// TIA Portal project "shift_registers" (V14)
// Cf. https://www.plctalk.net/qanda/showthread.php?t=128167

(* hardware
DEVICE "S7-1200 station_1"  S7-1200 Station
   slot 0: "Rack_0"  Rack  V1.0
   slot 1: "PLC_1"  CPU 1214C DC/DC/DC  6ES7 214-1AG40-0XB0  V4.2
DEVICE "HMI_1"  KTP700 Basic PN Portrait
   slot 0: "KTP700 Basic PN Portrait"  KTP700 Basic PN Portrait  6AV2 123-2GB03-0AX0  14.0.0.0
   slot 1: "HMI_RT_1"  KTP700 Basic PN Portrait  6AV2 123-2GB03-0AX0  14.0.0.0
   slot 5: "HMI_1.IE_CP_1"  PROFINET Interface  14.0.0.0
      slot 1: "PROFINET Interface_1"  PROFINET Interface
         slot 1: "Port_1"  Port
*)

// ===== PLC "PLC_1"  CPU 1214C DC/DC/DC =====

VAR_GLOBAL   // PLC tag table "Default tag table"
   "new_product_prox_input" AT %M0.6 : Bool;
   "HMI_ingest_input" AT %M0.7 : Bool;
   "HMI_target_line_input" AT %MW104 : Int;
   "HMI_target_pitch_input" AT %MW106 : Int;
   "Pause" AT %M1.1 : Bool;
   "current_pitch" AT %MW108 : Int;
   "valve_1" AT %M2.0 : Bool;
   "valve_2" AT %M2.1 : Bool;
   "valve_3" AT %M2.2 : Bool;
   "valve_4" AT %M2.3 : Bool;
   "valve_5" AT %M2.4 : Bool;
   "valve_6" AT %M2.5 : Bool;
   "Run" AT %M0.0 : Bool;
   "HMI_start_input" AT %M0.4 : Bool;
   "HMI_stop_input" AT %M0.5 : Bool;
   "pitch_prox_input" AT %M1.0 : Bool;
   "ingest_new" AT %M0.1 : Bool;
   "target_line" AT %MW100 : Int;
   "target_pitch" AT %MW102 : Int;
   "pitch_pulse" AT %M0.2 : Bool;
   "pitch_pulse_M" AT %M1.2 : Bool;
   "run_simulator" AT %M1.3 : Bool;
END_VAR

DATA_BLOCK "InputMap_DB"   // DB1
{ S7_Optimized_Access := 'TRUE' }
VERSION : 0.1
// stored: InstanceOfName InputMap
"InputMap"
BEGIN
END_DATA_BLOCK

DATA_BLOCK "LineValve_DB_1"   // DB2
{ S7_Optimized_Access := 'TRUE' }
VERSION : 0.1
// stored: InstanceOfName LineValve
"LineValve"
BEGIN
END_DATA_BLOCK

DATA_BLOCK "FIFO_BITS"   // DB3
{ S7_Optimized_Access := 'TRUE' }
VERSION : 0.1
   VAR
      fifo_bits : Array[0..511] of Byte;
   END_VAR
BEGIN
END_DATA_BLOCK

DATA_BLOCK "LineValve_DB_2"   // DB4
{ S7_Optimized_Access := 'TRUE' }
VERSION : 0.1
// stored: InstanceOfName LineValve
"LineValve"
BEGIN
END_DATA_BLOCK

DATA_BLOCK "LineValve_DB_3"   // DB5
{ S7_Optimized_Access := 'TRUE' }
VERSION : 0.1
// stored: InstanceOfName LineValve
"LineValve"
BEGIN
END_DATA_BLOCK

DATA_BLOCK "LineValve_DB_4"   // DB6
{ S7_Optimized_Access := 'TRUE' }
VERSION : 0.1
// stored: InstanceOfName LineValve
"LineValve"
BEGIN
END_DATA_BLOCK

DATA_BLOCK "LineValve_DB_5"   // DB7
{ S7_Optimized_Access := 'TRUE' }
VERSION : 0.1
// stored: InstanceOfName LineValve
"LineValve"
BEGIN
END_DATA_BLOCK

DATA_BLOCK "LineValve_DB_6"   // DB8
{ S7_Optimized_Access := 'TRUE' }
VERSION : 0.1
// stored: InstanceOfName LineValve
"LineValve"
BEGIN
END_DATA_BLOCK

DATA_BLOCK "Simulator_DB"   // DB9
{ S7_Optimized_Access := 'TRUE' }
VERSION : 0.1
// stored: InstanceOfName Simulator
"Simulator"
BEGIN
END_DATA_BLOCK

FUNCTION_BLOCK "InputMap"   // FB1, LAD
TITLE = Process HMI and sensor inputs
{ S7_Optimized_Access := 'TRUE' }
VERSION : 0.1
// N.B. new_product_prox_input probably needs a debounce for both 0-to-1 and 1-to-0 transitons; same for the pitch input
   VAR_INPUT
      new_product_prox_input : Bool;
      pitch_input : Bool;
   END_VAR
   VAR_OUTPUT
      Run_output : Bool;
      Pause_output : Bool;
      Ingest_output : Bool;
      target_line_output : Int;
      target_pitch_output : Int;
      pitch_pulse_output : Bool;
   END_VAR
   VAR_IN_OUT
      HMI_start_InOut : Bool;
      HMI_stop_InOut : Bool;
      HMI_ingest_InOut : Bool;
      HMI_target_line_InOut : Int;
      HMI_target_pitch_InOut : Int;
   END_VAR
   VAR
      Run : Bool;
      Pause : Bool;
      Ingest : Bool;
      new_product_prox_M : Bool;
      ingest_M : Bool;
      HMI_Line_pitch_offsets : Array[0..6] of Int;
   END_VAR
   VAR_TEMP   // added for the SCL form of the ladder/FBD networks
      _w1 : Bool;
      _w2 : Bool;
      _w3 : Bool;
   END_VAR
   // HMI_Line_pitch_offsets[1] := 4;
   // HMI_Line_pitch_offsets[2] := 8;
   // HMI_Line_pitch_offsets[3] := 12;
   // HMI_Line_pitch_offsets[4] := 16;
   // HMI_Line_pitch_offsets[5] := 20;
   // HMI_Line_pitch_offsets[6] := 24;
   // HMI_Line_pitch_offsets[0] := 0;
BEGIN

REGION Network 1: Process Start/Stop from HMI to Run
   // Also Reset HMI-driven Start/Stop to avoid anomalies if HMI does not return either of those momentaries to 0 ("set and forget")
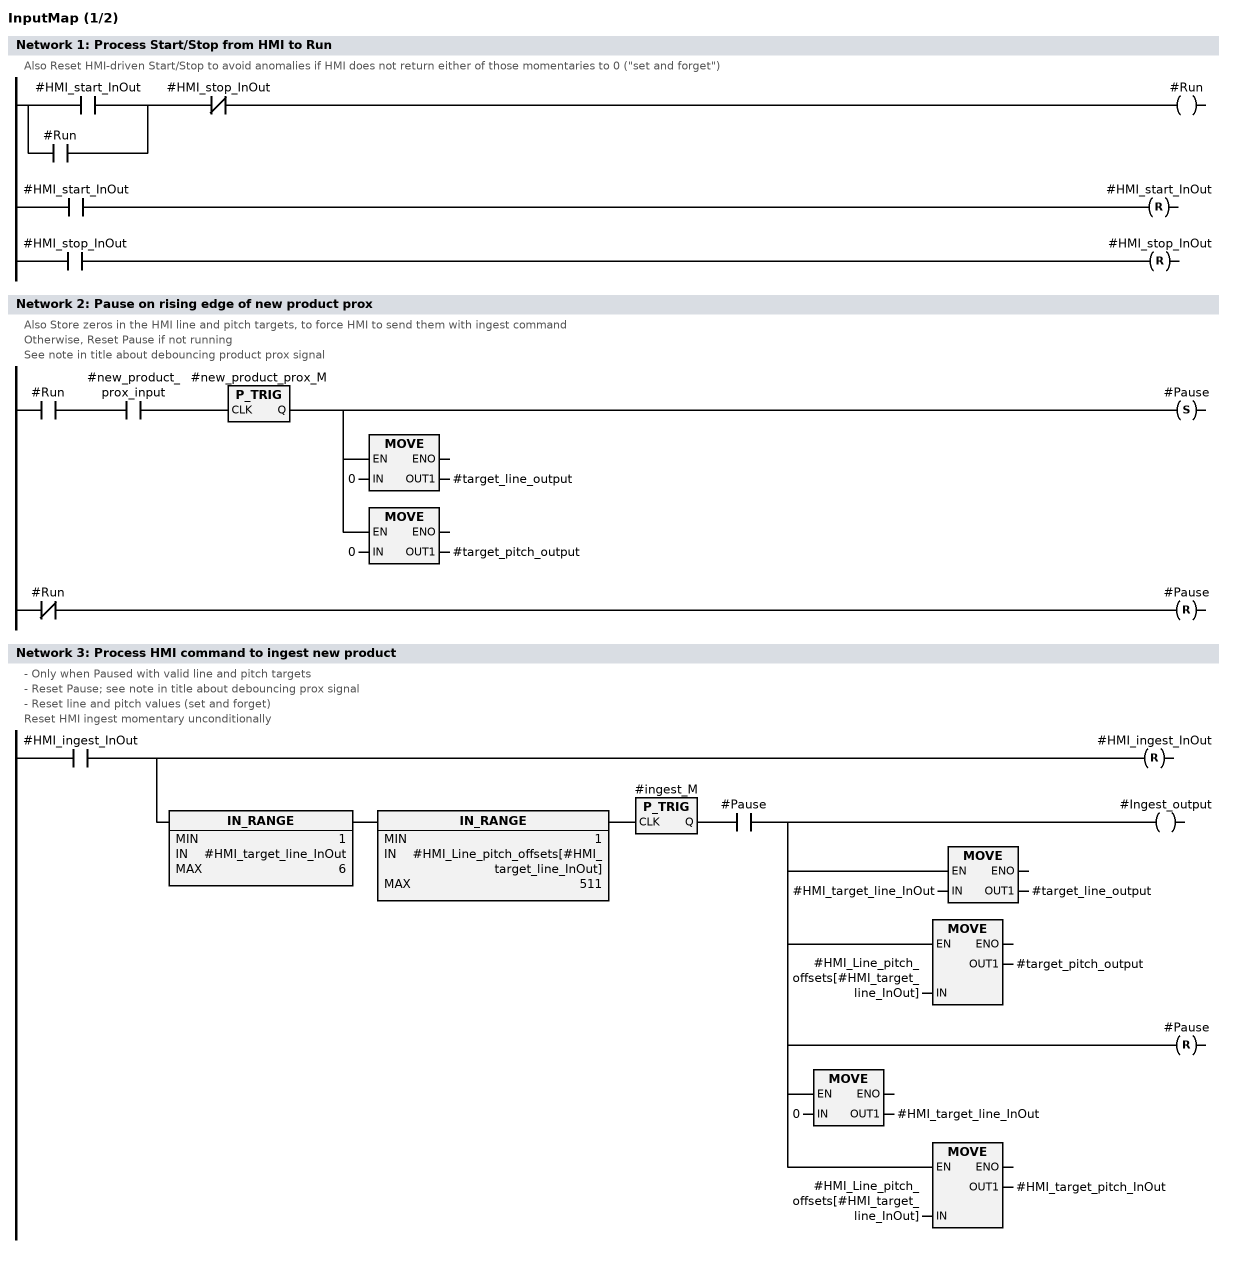
   RUNG wire#powerrail
      Contact( #HMI_start_InOut )
      wire#w1
      I_Contact( #HMI_stop_InOut )
      Coil( #Run )
   END_RUNG
   RUNG wire#powerrail
      Contact( #Run )
   END_RUNG wire#w1
   RUNG wire#powerrail
      Contact( #HMI_start_InOut )
      R_Coil( #HMI_start_InOut )
   END_RUNG
   RUNG wire#powerrail
      Contact( #HMI_stop_InOut )
      R_Coil( #HMI_stop_InOut )
   END_RUNG
   // the same network as SCL:
   #Run := (#HMI_start_InOut OR #Run) AND NOT #HMI_stop_InOut;
   IF #HMI_start_InOut THEN #HMI_start_InOut := FALSE; END_IF;
   IF #HMI_stop_InOut THEN #HMI_stop_InOut := FALSE; END_IF;
END_REGION

REGION Network 2: Pause on rising edge of new product prox
   // Also Store zeros in the HMI line and pitch targets, to force HMI to send them with ingest command
   // Otherwise, Reset Pause if not running
   // See note in title about debouncing product prox signal
   RUNG wire#powerrail
      Contact( #Run )
      Contact( #new_product_prox_input )
      P_Trig( #new_product_prox_M )
      wire#w1
      S_Coil( #Pause )
   END_RUNG
   RUNG wire#w1
      Move(in := 0, out1 => #target_line_output)
   END_RUNG
   RUNG wire#w1
      Move(in := 0, out1 => #target_pitch_output)
   END_RUNG
   RUNG wire#powerrail
      I_Contact( #Run )
      R_Coil( #Pause )
   END_RUNG
   // the same network as SCL:
   #_w1 := #Run AND #new_product_prox_input;
   #_w2 := #_w1 AND NOT #new_product_prox_M;   // rising edge
   #new_product_prox_M := #_w1;
   IF #_w2 THEN
       #Pause := TRUE;
       #target_line_output := 0;
       #target_pitch_output := 0;
   END_IF;
   IF NOT #Run THEN #Pause := FALSE; END_IF;
END_REGION

REGION Network 3: Process HMI command to ingest new product
   // - Only when Paused with valid line and pitch targets
   // - Reset Pause; see note in title about debouncing prox signal
   // - Reset line and pitch values (set and forget)
   // Reset HMI ingest momentary unconditionally
   RUNG wire#powerrail
      Contact( #HMI_ingest_InOut )
      wire#w1
      R_Coil( #HMI_ingest_InOut )
   END_RUNG
   RUNG wire#w1
      { S7_Templates := "SrcType := Int" } InRange(min := 1, in := #HMI_target_line_InOut, max := 6)
      { S7_Templates := "SrcType := Int" } InRange(min := 1, in := #HMI_Line_pitch_offsets[#HMI_target_line_InOut], max := 511)
      P_Trig( #ingest_M )
      Contact( #Pause )
      wire#w2
      Coil( #Ingest_output )
   END_RUNG
   RUNG wire#w2
      Move(in := #HMI_target_line_InOut, out1 => #target_line_output)
   END_RUNG
   RUNG wire#w2
      Move(in := #HMI_Line_pitch_offsets[#HMI_target_line_InOut], out1 => #target_pitch_output)
   END_RUNG
   RUNG wire#w2
      R_Coil( #Pause )
   END_RUNG
   RUNG wire#w2
      Move(in := 0, out1 => #HMI_target_line_InOut)
   END_RUNG
   RUNG wire#w2
      Move(in := #HMI_Line_pitch_offsets[#HMI_target_line_InOut], out1 => #HMI_target_pitch_InOut)
   END_RUNG
   // the same network as SCL:
   #_w1 := #HMI_ingest_InOut;
   IF #_w1 THEN #HMI_ingest_InOut := FALSE; END_IF;
   #_w2 := #_w1 AND (1 <= #HMI_target_line_InOut) AND (#HMI_target_line_InOut <= 6) AND (1 <= #HMI_Line_pitch_offsets[#HMI_target_line_InOut]) AND (#HMI_Line_pitch_offsets[#HMI_target_line_InOut] <= 511);
   #_w3 := #_w2 AND NOT #ingest_M;   // rising edge
   #ingest_M := #_w2;
   #Ingest_output := #_w3 AND #Pause;
   IF #Ingest_output THEN
       #target_line_output := #HMI_target_line_InOut;
       #target_pitch_output := #HMI_Line_pitch_offsets[#HMI_target_line_InOut];
       #Pause := FALSE;
       #HMI_target_line_InOut := 0;
       #HMI_target_pitch_InOut := #HMI_Line_pitch_offsets[#HMI_target_line_InOut];
   END_IF;
END_REGION

REGION Network 4: Push values to remaining outputs
   // - A debounce circuit for the pitch input might not go amiss here
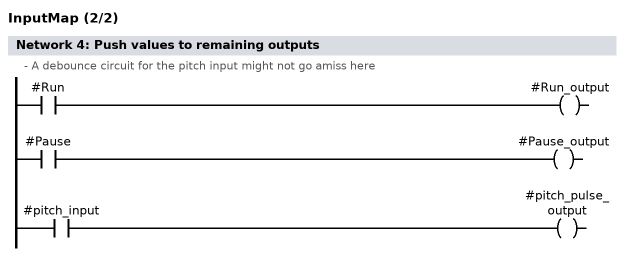
   RUNG wire#powerrail
      Contact( #Run )
      Coil( #Run_output )
   END_RUNG
   RUNG wire#powerrail
      Contact( #Pause )
      Coil( #Pause_output )
   END_RUNG
   RUNG wire#powerrail
      Contact( #pitch_input )
      Coil( #pitch_pulse_output )
   END_RUNG
   // the same network as SCL:
   #Run_output := #Run;
   #Pause_output := #Pause;
   #pitch_pulse_output := #pitch_input;
END_REGION
END_FUNCTION_BLOCK

FUNCTION_BLOCK "LineValve"   // FB2, LAD
TITLE = Process inputs for one Line-valve
{ S7_Optimized_Access := 'TRUE' }
VERSION : 0.1
// - Operate valve
// - Set up to ingest  three bits on ingest_pulse directed at this Line
// - Ingest those three bits on successive pitch rising edges
   VAR_INPUT
      target_line : Int;   // Line to ingest target_pitch if ingest_pulse is 0
      target_pitch : Int;   // Pitch offset of target_line if ingest_pulse is 0
      this_line : Int;   // Which Line this is
      current_pitch : Int;   // Conveyor start pitch offset into fifo_bits
      pitch_pulse : Bool;   // Pitch detection
   END_VAR
   VAR_OUTPUT
      operate_valve : Bool;   // Valve to direct product to ths Line
   END_VAR
   VAR_IN_OUT
      ingest_pulse : Bool;   // Bit commanding target_line to ingest target_pitch
      fifo_bits : Array[0..511] of Byte;   // Byte array containing product flag for all lines
   END_VAR
   VAR
      bits_to_ingest : Int;   // Remaining bits to ingest on pitch_pulse rising edges
      saved_pitch_offset : Int;   // Pitch offset from start of conveyor to this line's valve
      ingest_M : Bool;
   END_VAR
   VAR_TEMP
      this_bit_at_X7 : Byte;
      future_pitch : Int;
      this_bit : Int;
   END_VAR
   VAR CONSTANT
      pctX7 : Int := 2#10000000;
   END_VAR
   VAR_TEMP   // added for the SCL form of the ladder/FBD networks
      _w1 : Bool;
      _w2 : Bool;
   END_VAR
BEGIN

REGION Network 1: Operate valve when modeled product destined for this Line is near its Valve
   // Detect when the bit for this Line in Byte fifo_bits[current_pitch] is 1
   // - Bits in the static FIFO are cleared in Main [OB1] when current_pitch increments at pitch rising edge
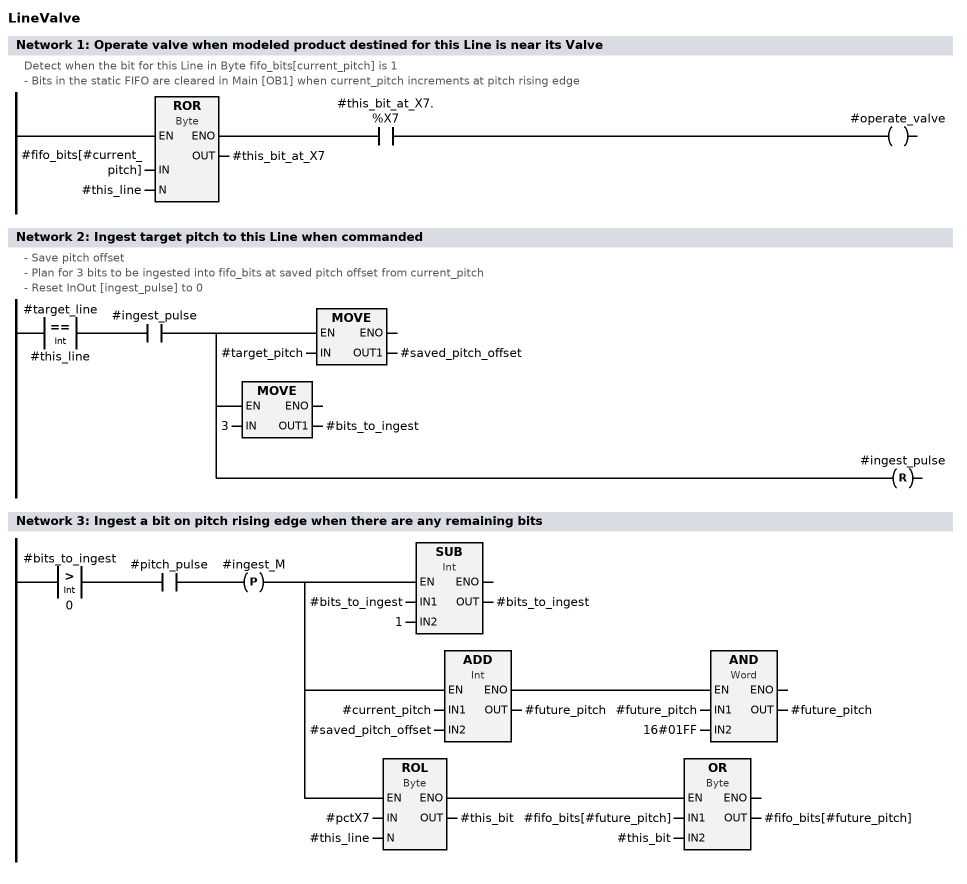
   #this_bit_at_X7 := ROR(IN := #fifo_bits[#current_pitch], N := #this_line);
   #operate_valve := #this_bit_at_X7.%X7;
END_REGION

REGION Network 2: Ingest target pitch to this Line when commanded
   // - Save pitch offset
   // - Plan for 3 bits to be ingested into fifo_bits at saved pitch offset from current_pitch
   // - Reset InOut [ingest_pulse] to 0
   RUNG wire#powerrail
      { S7_Templates := "SrcType := Int" } EQ_Contact(in1 := #target_line, in2 := #this_line)
      Contact( #ingest_pulse )
      wire#w1
      Move(in := #target_pitch, out1 => #saved_pitch_offset)
   END_RUNG
   RUNG wire#w1
      Move(in := 3, out1 => #bits_to_ingest)
   END_RUNG
   RUNG wire#w1
      R_Coil( #ingest_pulse )
   END_RUNG
   // the same network as SCL:
   IF (#target_line = #this_line) AND #ingest_pulse THEN
       #saved_pitch_offset := #target_pitch;
       #bits_to_ingest := 3;
       #ingest_pulse := FALSE;
   END_IF;
END_REGION

REGION Network 3: Ingest a bit on pitch rising edge when there are any remaining bits
   // no checked SCL form for this network; see the picture
END_REGION
END_FUNCTION_BLOCK

FUNCTION_BLOCK "Simulator"   // FB3, LAD
TITLE = Model/simulate synthetic inputs from HMI and physical sensors (pitch and new product proxes)
{ S7_Optimized_Access := 'TRUE' }
VERSION : 0.1
   VAR_INPUT
      Run_this_sim_Input : Bool;
      Run_Input : Bool;
      Pause_Input : Bool;
   END_VAR
   VAR_IN_OUT
      pitch_prox_InOut : Bool;
      new_product_prox_InOut : Bool;
   END_VAR
   VAR
      time_status : Int;
      time_dtl : DTL;
      next_target_line : Int;
      IEC_prox_delay : IEC_TIMER;
      second : USInt;
      nanosecond : UDInt;
      two_second_M : Bool;
      prox_pulse : Bool;
      new_product_prox_delay_count : Int;
   END_VAR
   VAR_TEMP   // added for the SCL form of the ladder/FBD networks
      _w1 : Bool;
      _w2 : Bool;
      _w3 : Bool;
   END_VAR
BEGIN

REGION Network 1: RETurn if simulator is not to be run
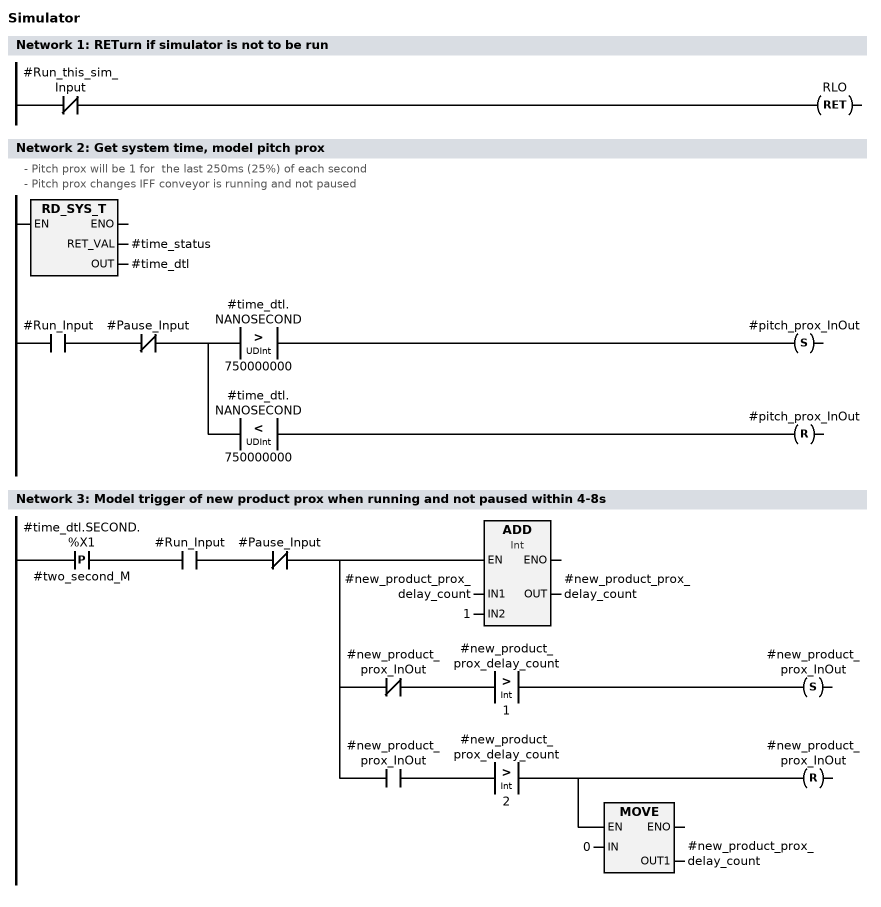
   IF NOT #Run_this_sim_Input THEN
       ENO := TRUE;
       RETURN;
   END_IF;
END_REGION

REGION Network 2: Get system time, model pitch prox
   // - Pitch prox will be 1 for  the last 250ms (25%) of each second
   // - Pitch prox changes IFF conveyor is running and not paused
   #time_status := RD_SYS_T(OUT => #time_dtl);
   #_w1 := #Run_Input AND NOT #Pause_Input;
   IF #_w1 AND (#time_dtl.NANOSECOND > 750000000) THEN #pitch_prox_InOut := TRUE; END_IF;
   IF #_w1 AND (#time_dtl.NANOSECOND < 750000000) THEN #pitch_prox_InOut := FALSE; END_IF;
END_REGION

REGION Network 3: Model trigger of new product prox when running and not paused within 4-8s
   RUNG wire#powerrail
      P_Contact(operand := #time_dtl.SECOND.%X1, bit := #two_second_M)
      Contact( #Run_Input )
      I_Contact( #Pause_Input )
      wire#w1
      { S7_Templates := "SrcType := Int" } Add(in1 := #new_product_prox_delay_count, in2 := 1, out => #new_product_prox_delay_count)
   END_RUNG
   RUNG wire#w1
      I_Contact( #new_product_prox_InOut )
      { S7_Templates := "SrcType := Int" } GT_Contact(in1 := #new_product_prox_delay_count, in2 := 1)
      S_Coil( #new_product_prox_InOut )
   END_RUNG
   RUNG wire#w1
      Contact( #new_product_prox_InOut )
      { S7_Templates := "SrcType := Int" } GT_Contact(in1 := #new_product_prox_delay_count, in2 := 2)
      wire#w2
      R_Coil( #new_product_prox_InOut )
   END_RUNG
   RUNG wire#w2
      Move(in := 0, out1 => #new_product_prox_delay_count)
   END_RUNG
   // the same network as SCL:
   #_w1 := #time_dtl.SECOND.%X1 AND NOT #two_second_M;   // rising edge of #time_dtl.SECOND.%X1
   #two_second_M := #time_dtl.SECOND.%X1;
   #_w2 := #_w1 AND #Run_Input AND NOT #Pause_Input;
   IF #_w2 THEN #new_product_prox_delay_count := #new_product_prox_delay_count + 1; END_IF;
   IF #_w2 AND NOT #new_product_prox_InOut AND (#new_product_prox_delay_count > 1) THEN
       #new_product_prox_InOut := TRUE;
   END_IF;
   #_w3 := #_w2 AND #new_product_prox_InOut AND (#new_product_prox_delay_count > 2);
   IF #_w3 THEN
       #new_product_prox_InOut := FALSE;
       #new_product_prox_delay_count := 0;
   END_IF;
END_REGION
END_FUNCTION_BLOCK

ORGANIZATION_BLOCK "Main"   // OB1, LAD, ProgramCycle
TITLE = "Main Program Sweep (Cycle)"
{ S7_Optimized_Access := 'TRUE' }
VERSION : 0.1
   VAR_INPUT
      Initial_Call : Bool;   // Initial call of this OB
      Remanence : Bool;   // =True, if remanent data are available
   END_VAR
   VAR_TEMP   // added for the SCL form of the ladder/FBD networks
      _w1 : Bool;
      _w2 : Bool;
      _w3 : Bool;
   END_VAR
BEGIN

REGION Network 1
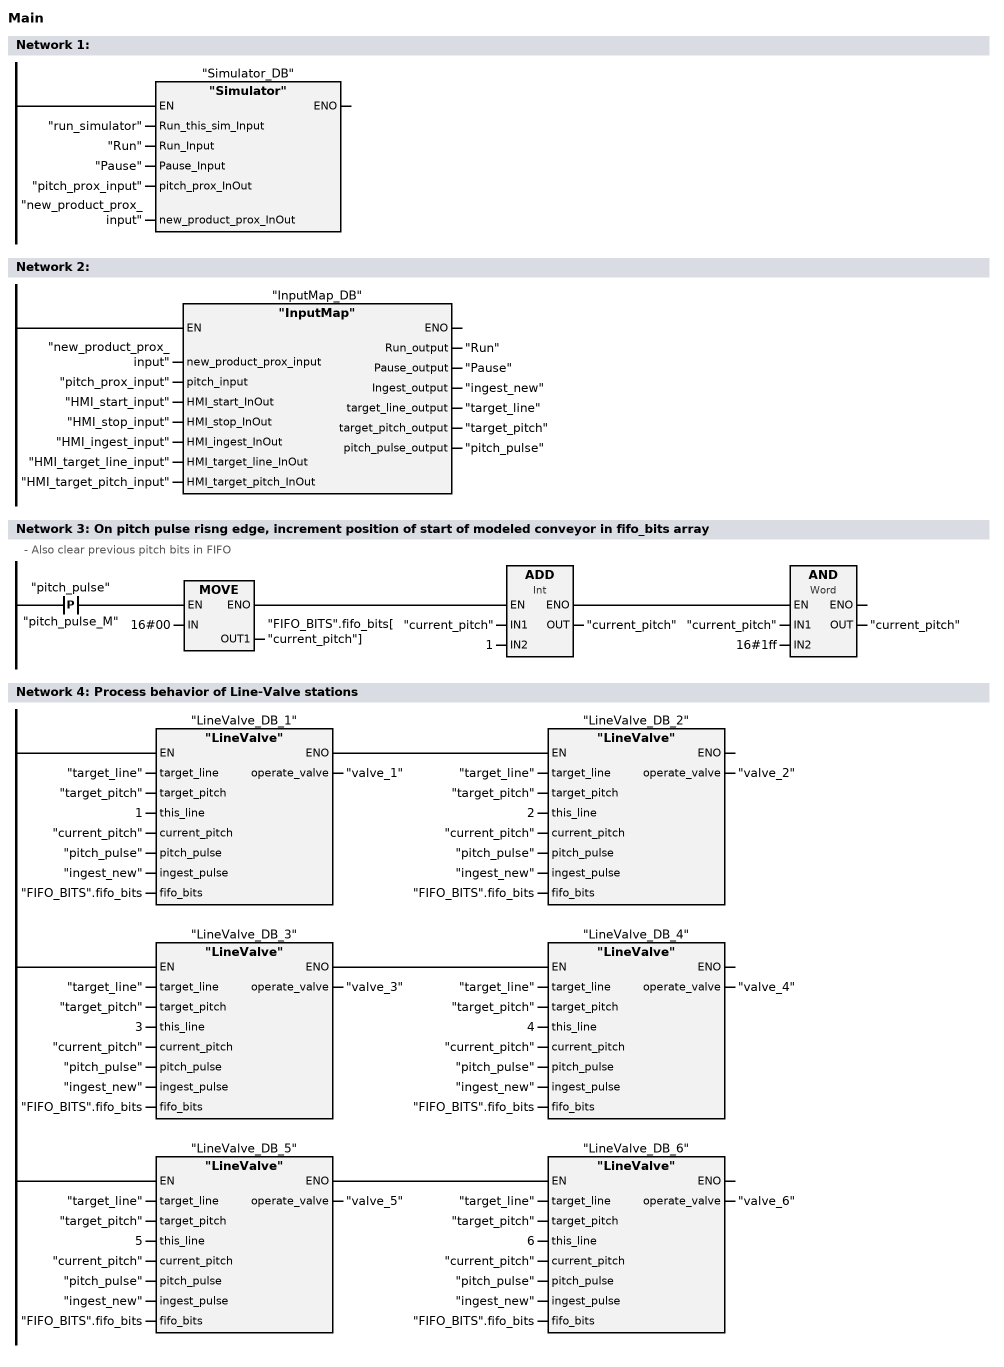
   RUNG wire#powerrail
      "Simulator_DB"(Run_this_sim_Input := "run_simulator", Run_Input := "Run", Pause_Input := "Pause", pitch_prox_InOut := "pitch_prox_input", new_product_prox_InOut := "new_product_prox_input")
   END_RUNG
   // the same network as SCL:
   "Simulator_DB"(Run_this_sim_Input := "run_simulator",   // "Simulator"
                  Run_Input := "Run",
                  Pause_Input := "Pause",
                  pitch_prox_InOut := "pitch_prox_input",
                  new_product_prox_InOut := "new_product_prox_input");
END_REGION

REGION Network 2
   RUNG wire#powerrail
      "InputMap_DB"(new_product_prox_input := "new_product_prox_input", pitch_input := "pitch_prox_input", HMI_start_InOut := "HMI_start_input", HMI_stop_InOut := "HMI_stop_input", HMI_ingest_InOut := "HMI_ingest_input", HMI_target_line_InOut := "HMI_target_line_input", HMI_target_pitch_InOut := "HMI_target_pitch_input", Run_output => "Run", Pause_output => "Pause", Ingest_output => "ingest_new", target_line_output => "target_line", target_pitch_output => "target_pitch", pitch_pulse_output => "pitch_pulse")
   END_RUNG
   // the same network as SCL:
   "InputMap_DB"(new_product_prox_input := "new_product_prox_input",   // "InputMap"
                 pitch_input := "pitch_prox_input",
                 HMI_start_InOut := "HMI_start_input",
                 HMI_stop_InOut := "HMI_stop_input",
                 HMI_ingest_InOut := "HMI_ingest_input",
                 HMI_target_line_InOut := "HMI_target_line_input",
                 HMI_target_pitch_InOut := "HMI_target_pitch_input",
                 Run_output => "Run",
                 Pause_output => "Pause",
                 Ingest_output => "ingest_new",
                 target_line_output => "target_line",
                 target_pitch_output => "target_pitch",
                 pitch_pulse_output => "pitch_pulse");
END_REGION

REGION Network 3: On pitch pulse risng edge, increment position of start of modeled conveyor in fifo_bits array
   // - Also clear previous pitch bits in FIFO
   // no checked SCL form for this network; see the picture
END_REGION

REGION Network 4: Process behavior of Line-Valve stations
   RUNG wire#powerrail
      "LineValve_DB_1"(target_line := "target_line", target_pitch := "target_pitch", this_line := 1, current_pitch := "current_pitch", pitch_pulse := "pitch_pulse", ingest_pulse := "ingest_new", fifo_bits := "FIFO_BITS".fifo_bits, operate_valve => "valve_1")
      "LineValve_DB_2"(target_line := "target_line", target_pitch := "target_pitch", this_line := 2, current_pitch := "current_pitch", pitch_pulse := "pitch_pulse", ingest_pulse := "ingest_new", fifo_bits := "FIFO_BITS".fifo_bits, operate_valve => "valve_2")
   END_RUNG
   RUNG wire#powerrail
      "LineValve_DB_3"(target_line := "target_line", target_pitch := "target_pitch", this_line := 3, current_pitch := "current_pitch", pitch_pulse := "pitch_pulse", ingest_pulse := "ingest_new", fifo_bits := "FIFO_BITS".fifo_bits, operate_valve => "valve_3")
      "LineValve_DB_4"(target_line := "target_line", target_pitch := "target_pitch", this_line := 4, current_pitch := "current_pitch", pitch_pulse := "pitch_pulse", ingest_pulse := "ingest_new", fifo_bits := "FIFO_BITS".fifo_bits, operate_valve => "valve_4")
   END_RUNG
   RUNG wire#powerrail
      "LineValve_DB_5"(target_line := "target_line", target_pitch := "target_pitch", this_line := 5, current_pitch := "current_pitch", pitch_pulse := "pitch_pulse", ingest_pulse := "ingest_new", fifo_bits := "FIFO_BITS".fifo_bits, operate_valve => "valve_5")
      "LineValve_DB_6"(target_line := "target_line", target_pitch := "target_pitch", this_line := 6, current_pitch := "current_pitch", pitch_pulse := "pitch_pulse", ingest_pulse := "ingest_new", fifo_bits := "FIFO_BITS".fifo_bits, operate_valve => "valve_6")
   END_RUNG
   // the same network as SCL:
   "LineValve_DB_1"(target_line := "target_line",   // "LineValve"
                    target_pitch := "target_pitch",
                    this_line := 1,
                    current_pitch := "current_pitch",
                    pitch_pulse := "pitch_pulse",
                    ingest_pulse := "ingest_new",
                    fifo_bits := "FIFO_BITS".fifo_bits,
                    operate_valve => "valve_1",
                    ENO => #_w1);
   IF #_w1 THEN
       "LineValve_DB_2"(target_line := "target_line",   // "LineValve"
                        target_pitch := "target_pitch",
                        this_line := 2,
                        current_pitch := "current_pitch",
                        pitch_pulse := "pitch_pulse",
                        ingest_pulse := "ingest_new",
                        fifo_bits := "FIFO_BITS".fifo_bits,
                        operate_valve => "valve_2");
   END_IF;
   "LineValve_DB_3"(target_line := "target_line",   // "LineValve"
                    target_pitch := "target_pitch",
                    this_line := 3,
                    current_pitch := "current_pitch",
                    pitch_pulse := "pitch_pulse",
                    ingest_pulse := "ingest_new",
                    fifo_bits := "FIFO_BITS".fifo_bits,
                    operate_valve => "valve_3",
                    ENO => #_w2);
   IF #_w2 THEN
       "LineValve_DB_4"(target_line := "target_line",   // "LineValve"
                        target_pitch := "target_pitch",
                        this_line := 4,
                        current_pitch := "current_pitch",
                        pitch_pulse := "pitch_pulse",
                        ingest_pulse := "ingest_new",
                        fifo_bits := "FIFO_BITS".fifo_bits,
                        operate_valve => "valve_4");
   END_IF;
   "LineValve_DB_5"(target_line := "target_line",   // "LineValve"
                    target_pitch := "target_pitch",
                    this_line := 5,
                    current_pitch := "current_pitch",
                    pitch_pulse := "pitch_pulse",
                    ingest_pulse := "ingest_new",
                    fifo_bits := "FIFO_BITS".fifo_bits,
                    operate_valve => "valve_5",
                    ENO => #_w3);
   IF #_w3 THEN
       "LineValve_DB_6"(target_line := "target_line",   // "LineValve"
                        target_pitch := "target_pitch",
                        this_line := 6,
                        current_pitch := "current_pitch",
                        pitch_pulse := "pitch_pulse",
                        ingest_pulse := "ingest_new",
                        fifo_bits := "FIFO_BITS".fifo_bits,
                        operate_valve => "valve_6");
   END_IF;
END_REGION
END_ORGANIZATION_BLOCK

(* ===== HMI "HMI_RT_1" =====
system functions are stored by id; their names below are inferred from use
connection "HMI_Connection_1": ETHERNET, SMART_S7_1200_OMS

HMI tags "Default tag table"
   "HMI_Line_1_pitch_offset" : Int = PLC InputMap_DB.HMI_Line_pitch_offsets[1] AT %DB1.DBW0, 1 s
   "HMI_Line_2_pitch_offset" : Int = PLC InputMap_DB.HMI_Line_pitch_offsets[2] AT %DB1.DBW0, 1 s
   "HMI_Line_3_pitch_offset" : Int = PLC InputMap_DB.HMI_Line_pitch_offsets[3] AT %DB1.DBW0, 1 s
   "HMI_Line_4_pitch_offset" : Int = PLC InputMap_DB.HMI_Line_pitch_offsets[4] AT %DB1.DBW0, 1 s
   "HMI_Line_5_pitch_offset" : Int = PLC InputMap_DB.HMI_Line_pitch_offsets[5] AT %DB1.DBW0, 1 s
   "HMI_Line_6_pitch_offset" : Int = PLC InputMap_DB.HMI_Line_pitch_offsets[6] AT %DB1.DBW0, 1 s
   "HMI_target_pitch_input_mux" : Int, internal
   "HMI_target_line_input" : Int = PLC HMI_target_line_input AT %MW104, 1 s
   "HMI_Line" : Int, internal
   "HMI_target_pitch_input" : Int = PLC HMI_target_pitch_input AT %MW106, 1 s
   "HMI_Line_0_pitch_offset" : Int = PLC InputMap_DB.HMI_Line_pitch_offsets[0] AT %DB1.DBW0, 1 s
   "HMI_ingest_input" : Bool = PLC HMI_ingest_input AT %M0.7, 1 s
   "HMI_start_input" : Bool = PLC HMI_start_input AT %M0.4, 1 s
   "HMI_stop_input" : Bool = PLC HMI_stop_input AT %M0.5, 1 s
   "Pause" : Bool = PLC Pause AT %M1.1, 1 s
   "Run" : Bool = PLC Run AT %M0.0, 1 s
   "valve_1" : Bool = PLC valve_1 AT %M2.0, 1 s
   "valve_2" : Bool = PLC valve_2 AT %M2.1, 1 s
   "valve_3" : Bool = PLC valve_3 AT %M2.2, 1 s
   "valve_4" : Bool = PLC valve_4 AT %M2.3, 1 s
   "valve_5" : Bool = PLC valve_5 AT %M2.4, 1 s
   "valve_6" : Bool = PLC valve_6 AT %M2.5, 1 s
   "current_pitch" : Int = PLC current_pitch AT %MW108, 1 s

screen "Screen_1" 480x800
   Button "Button_1" at 24,16 size 100x40; TextOff 'Start'
      on Press: SetTag("HMI_start_input", 1)
   Button "Button_2" at 360,16 size 93x39; TextOff 'Stop'
      on Press: SetTag("HMI_stop_input", 1)
   IOField "I/O field_1" at 26,115 size 48x40; HelpText 'Pitch offset for Line-Valve 1'; FormatPattern 999
      ProcessValue <- "HMI_Line_1_pitch_offset"
   Ellipse "Ellipse_1" at 256,161 size 48x48
      Appearance <- "Pause"
   TextField "Text field_1" at 248,97 size 70x61; Text 'Paused; Product Present'
   Button "Button_3" at 83,115 size 112x40; TextOff 'Line-Valve 1'; HelpText 'Press to stage [pitch offset] and [Line Number] for sending to controller for current new product'
      on Click: SetTag("HMI_target_line_input", 1)
   IOField "I/O field_2" at 26,163 size 48x40; HelpText 'Pitch offset for Line-Valve 2'; FormatPattern 999
      ProcessValue <- "HMI_Line_2_pitch_offset"
   Button "Button_4" at 83,163 size 112x40; TextOff 'Line-Valve 2'; HelpText 'Press to stage [pitch offset] and [Line Number] for sending to controller for current new product'
      on Click: SetTag("HMI_target_line_input", 2)
   IOField "I/O field_3" at 26,211 size 48x40; HelpText 'Pitch offset for Line-Valve 3'; FormatPattern 999
      ProcessValue <- "HMI_Line_3_pitch_offset"
   Button "Button_5" at 83,211 size 112x40; TextOff 'Line-Valve 3'; HelpText 'Press to stage [pitch offset] and [Line Number] for sending to controller for current new product'
      on Click: SetTag("HMI_target_line_input", 3)
   IOField "I/O field_4" at 26,259 size 48x40; HelpText 'Pitch offset for Line-Valve 4'; FormatPattern 999
      ProcessValue <- "HMI_Line_4_pitch_offset"
   Button "Button_6" at 83,259 size 112x40; TextOff 'Line-Valve 4'; HelpText 'Press to stage [pitch offset] and [Line Number] for sending to controller for current new product'
      on Click: SetTag("HMI_target_line_input", 4)
   IOField "I/O field_5" at 26,307 size 48x40; HelpText 'Pitch offset for Line-Valve 5'; FormatPattern 999
      ProcessValue <- "HMI_Line_5_pitch_offset"
   Button "Button_7" at 83,307 size 112x40; TextOff 'Line-Valve 5'; HelpText 'Press to stage [pitch offset] and [Line Number] for sending to controller for current new product'
      on Click: SetTag("HMI_target_line_input", 5)
   IOField "I/O field_6" at 26,355 size 48x40; HelpText 'Pitch offset for Line-Valve 6'; FormatPattern 999
      ProcessValue <- "HMI_Line_6_pitch_offset"
   Button "Button_8" at 83,355 size 112x40; TextOff 'Line-Valve 6'; HelpText 'Press to stage [pitch offset] and [Line Number] for sending to controller for current new product'
      on Click: SetTag("HMI_target_line_input", 6)
   IOField "I/O field_7" at 224,235 size 48x40; HelpText 'Pitch offset for sending to controller for current new product'; FormatPattern 999
      ProcessValue <- "HMI_target_pitch_input_mux"
   IOField "I/O field_8" at 296,234 size 48x40; HelpText 'Pitch offset for sending to controller for current new product'; FormatPattern 9
      ProcessValue <- "HMI_target_line_input"
   Button "Button_9" at 224,280 size 120x48; TextOff 'Direct New Product'
      on Press: SetTag("HMI_ingest_input", 1)
   Ellipse "Ellipse_2" at 192,8 size 48x48
      Appearance <- "Run"
   Ellipse "Ellipse_3" at 416,112 size 48x48
      Appearance <- "valve_1"
   Ellipse "Ellipse_4" at 416,160 size 48x48
      Appearance <- "valve_2"
   Ellipse "Ellipse_5" at 416,207 size 48x48
      Appearance <- "valve_3"
   Ellipse "Ellipse_6" at 416,254 size 48x48
      Appearance <- "valve_4"
   Ellipse "Ellipse_7" at 416,301 size 48x48
      Appearance <- "valve_5"
   Ellipse "Ellipse_8" at 416,348 size 48x48
      Appearance <- "valve_6"
   IOField "I/O field_9" at 224,360 size 120x40; FormatPattern 999
      ProcessValue <- "current_pitch"
   TextField "Text field_2" at 408,80 size 58x23; Text 'Valves'
   TextField "Text field_3" at 26,91 size 46x23; Text 'Pitch'
   TextField "Text field_4" at 99,70 size 83x42; Text 'Load Line and Pitch'
   TextField "Text field_5" at 224,336 size 112x23; Text 'Current pitch'
   TextField "Text field_6" at 225,211 size 46x23; Text 'Pitch'
   TextField "Text field_7" at 299,211 size 39x23; Text 'Line'
   TextField "Text field_8" at 241,20 size 72x23; Text 'Running'
*)